FUNCTION_BLOCK DFB_FacilityAlarm_1
VAR_INPUT
	Sec_P					: BOOL; // Second pulse
	TbotNo					: INT; // 1: Tbot left, 2: Tbot right
	PV						: LREAL; // Process Value
	WarningTimer			: UDINT;
	AlarmTimer				: UDINT;
	AbortTimer				: UDINT;
	DB						: LREAL	:= 0.2; // Deadband
	LogName					: STRING;
	ModuleID				: E_ModuleID;
	EventName				: E_EventName;
END_VAR

VAR_OUTPUT
	Warning					: BOOL;
	Alarm					: BOOL;
	Abort					: BOOL;
END_VAR

VAR_IN_OUT
	LowSP					: LREAL; // Low Alarm Set Point
	LowLowSP				: LREAL; // Low Low Alarm Set Point
END_VAR

VAR
	_State_Changed			: BOOL;
	
	_State					: INT;
	_Last_State				: INT;
	_TLast_State			: INT;
	
	_State_Timer			: UDINT;
	
	
	_EmptyEvent				: ST_Event;
	
	_TON_Warning			: TON;
	_TON_Alarm				: TON;		
END_VAR

///////////////////////////////////////////////////////////////////////////////////////////////////////////////////////////////////////////////////////////////////////////////
//	State timer
///////////////////////////////////////////////////////////////////////////////////////////////////////////////////////////////////////////////////////////////////////////////

_State_Changed									:= _State <> _TLast_State;
_TLast_State									:= _State;

IF _State_Changed THEN
	_State_Timer								:= 0;
	Logging.fbDebugLog.M_nLogger(iLogLevel:= iLogVerbosity, sSource:= 'AIN Log', 
		sMessage								:= CONCAT(CONCAT(LogName, 'current state['),
														 CONCAT(INT_TO_STRING(_State), ']'))); 
	
ELSE
	IF Sec_P THEN
		_State_Timer							:= _State_Timer + 1;
	END_IF
END_IF


///////////////////////////////////////////////////////////////////////////////////////////////////////////////////////////////////////////////////////////////////////////////
//	Safety clamp
///////////////////////////////////////////////////////////////////////////////////////////////////////////////////////////////////////////////////////////////////////////////

IF LowSP < LowLowSP THEN
	LowSP										:= LowLowSP;
END_IF

///////////////////////////////////////////////////////////////////////////////////////////////////////////////////////////////////////////////////////////////////////////////
//	State case
///////////////////////////////////////////////////////////////////////////////////////////////////////////////////////////////////////////////////////////////////////////////

CASE _State OF
	0: (*Idle*)
	
		(*Action*)
		Warning									:= FALSE;
		Alarm									:= FALSE;
		Abort									:= FALSE;
		_TON_Warning(IN:= FALSE, PT:= UDINT_TO_TIME(WarningTimer * 1000));
		
		(*Transition*)
		IF PV < LowLowSP THEN
			_TON_Warning(IN:= TRUE, PT:= UDINT_TO_TIME(WarningTimer * 1000));
			_State								:= 21; // Low Low Alarm - Delay
		ELSIF PV < LowSP THEN
			_TON_Warning(IN:= TRUE, PT:= UDINT_TO_TIME(WarningTimer * 1000));
			_State								:= 11; // Low Alarm - Delay
		END_IF
		
	11: (*Low Alarm - Delay*)
		_Last_State								:= 11;
		
		(*Action*)
		Warning									:= TRUE;
		Alarm									:= FALSE;
		Abort									:= FALSE;
		
		(*Transition*)
		IF PV >= LowSP + DB THEN
			_State								:= 0; // Idle
		ELSIF PV < LowLowSP THEN
			_State								:= 21; // Low Low Alarm - Delay
		ELSIF _State_Timer >= WarningTimer THEN
			_State								:= 22; // Low Alarm - Send Event
		END_IF
	
	21: (*Low Low Alarm - Delay*)
		_Last_State								:= 21;
		
		(*Action*)
		Warning									:= FALSE;
		Alarm									:= TRUE;
		Abort									:= FALSE;
		
		(*Transition*)
		IF PV >= LowSP + DB THEN
			_State								:= 0; // Idle
		ELSIF _State_Timer >= AlarmTimer THEN
			_State								:= 24; // Low Low Alarm - Send Event
		END_IF
	
	22:	(*Low Alarm - Send Event*)
		_Last_State								:= 22;
		
		(*Action*)
		Warning									:= TRUE;
		Alarm									:= FALSE;
		Abort									:= FALSE;
		
		// Event - AbortInProgress
		CmdAndEventProcess.fbCmdAndEventUpdate.M_AddEvent(
			sLogName							:= LogName, 
			eEventName							:= EventName, 
			eModuleID							:= ModuleID, 
			iParam								:= _EmptyEvent.iParam,
			sParam								:= _EmptyEvent.sParam, 
			bParam								:= _EmptyEvent.bParam, 
			dParam								:= _EmptyEvent.dParam,
			sFailReason							:= '');
		
		(*Transition*)
		_State									:= 25; // Low Alarm - Check abort time
		
	24: (*Low Low Alarm - Send Event*)
		_Last_State								:= 24;
		
		(*Action*)
		Warning									:= FALSE;
		Alarm									:= TRUE;
		Abort									:= FALSE;
		
		// Event - AbortInProgress
		CmdAndEventProcess.fbCmdAndEventUpdate.M_AddEvent(
			sLogName							:= LogName, 
			eEventName							:= EventName, 
			eModuleID							:= ModuleID, 
			iParam								:= _EmptyEvent.iParam,
			sParam								:= _EmptyEvent.sParam, 
			bParam								:= _EmptyEvent.bParam, 
			dParam								:= _EmptyEvent.dParam,
			sFailReason							:= '');
		
		(*Transition*)
		_State									:= 26; // Low Low Alarm - Check abort time
		
	25: (*Low Alarm - Check abort time*)
		_Last_State								:= 25;
		
		(*Action*)
		Warning									:= TRUE;
		Alarm									:= FALSE;
		Abort									:= FALSE;
		
		(*Transition*)
		IF _State_Timer >= AbortTimer THEN
			_State								:= 40; // Abort
		END_IF
		
	26: (*Low Low Alarm - Check abort time*)
		_Last_State								:= 26;
		
		(*Action*)
		Warning									:= TRUE;
		Alarm									:= TRUE;
		Abort									:= FALSE;
		
		(*Transition*)
		IF _State_Timer >= AbortTimer THEN
			_State								:= 41; // Abort
		(*ELSIF PV >= LowLowSP + DB THEN
			_State								:= 21; // Low Low Alarm - Delay
		ELSIF PV >= LowSP + DB THEN
			_State								:= 11; // Low Alarm - Delay*)
		END_IF
		
	40: (*Abort*)
		_Last_State								:= 40;
		
		(*Action*)
		Warning									:= TRUE;
		Alarm									:= FALSE;
		Abort									:= TRUE;
		
		(*Transition*)
		IF PV >= LowSP + DB THEN
			_State								:= 0; // Idle
		END_IF
		
	41: (*Abort*)
		_Last_State								:= 41;
		
		(*Action*)
		Warning									:= TRUE;
		Alarm									:= TRUE;
		Abort									:= TRUE;
		
		(*Transition*)
		IF PV >= LowSP + DB THEN
			_State								:= 0; // Idle
		END_IF
END_CASE

END_FUNCTION_BLOCK

(* stored: Version 1.1.0.1, ProductVersion 3.1.4022.18
   POU DFB_FacilityAlarm_1: Id {3342c78a-600c-4bb8-80f5-0ed514ce7eee}, SpecialFunc None *)
